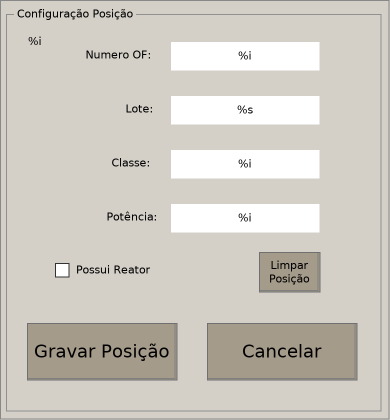
VISUALIZATION ConfigPosicao  // 390x420
VAR_IN_OUT
	bReator: BOOL;
	iOFnumber: INT;
	iSrlNumber: INT;
	
	
	
END_VAR
    GroupBox (6,6 375x405), "Configuração Posição"
        Checkbox (47,251 110x26), "Possui Reator", variable: gravarConfigPosicao.bReator[GVL.actEst]
        Label (72,34 81x30), "Numero OF:"
        Textfield (164,35 150x30), "%i", text variable: GVL.cfgPos_OF019
            OnMouseDown: write the text variable via VisuDialogs.Numpad
        Label (42,88 108x30), "Lote:"
        Textfield (164,89 150x30), "%s", text variable: GVL.cfgPos_LT019
            OnMouseDown: write the text variable via VisuDialogs.Keypad
        Label (97,142 56x30), "Classe:"
        Button (21,317 150x57), "Gravar Posição"
            OnMouseClick: CloseDialog Dialog=ConfigPosicao, Result=OK, NumpadKeypadSet=True
            OnMouseClick: execute { gravarConfigPosicao(); }
        Button (201,317 150x57), "Cancelar"
            OnMouseClick: CloseDialog Dialog=ConfigPosicao, Result=Cancel, NumpadKeypadSet=True
        Button (253,246 61x40), "Limpar Posição"
            OnMouseClick: CloseDialog Dialog=ConfigPosicao, Result=Cancel, NumpadKeypadSet=True
            OnMouseClick: execute {
                gvl_p.aPositionsE019[gvl.actPos].numOF:='0';
                gvl_p.aPositionsE019[gvl.actPos].lote:='0';
                gvl_p.aPositionsE019[gvl.actPos].class:=0;
                gvl_p.aPositionsE019[gvl.actPos].pot:=0;
                gvl_p.aPositionsE019[gvl.actPos].cor:=0;
                IF gvl.totalPos[gvl.actEst] <> 0 THEN
                gvl.totalPos[gvl.actEst]:= gvl.totalPos[gvl.actEst] - 1;
                ELSE
                	gvl.totalPos[gvl.actEst] := 0;
                END_IF
                gravarConfigPosicao.bReator[0]:= false;
                ///// GERADOR DE LOG -------------------------------------------------------------
                gvl.envialog:= 'Posição Nº ';
                gvl.envialog:= concat(gvl.envialog, INT_TO_STRING(gvl.actPos));
                gvl.envialog:= concat(gvl.envialog,' foi limpa. ESTUFA ');
                gvl.envialog:= concat(gvl.envialog, INT_TO_STRING(gvl.actEst));
                gvl.logRegister[gvl.actEst]:= gvl.envialog;
            }
        Textfield (164,143 150x30), "%i", text variable: GVL.cfgPos_Class019
            OnMouseDown: write the text variable via VisuDialogs.Numpad
        Textfield (164,197 150x30), "%i", text variable: GVL.cfgPos_Pot019
            OnMouseDown: write the text variable via VisuDialogs.Numpad
    Label (104,202 56x30), "Potência:"
    Rectangle (24,30 22x23), "%i", text variable: GVL.actPos
END_VISUALIZATION

(* stored: Version 1.1.0.1, ProductVersion 3.1.4024.12
   Visu ConfigPosicao: Id {a6174f95-717c-4e04-bf54-2d0ebd257176} *)
